FUNCTION "JsonW_LNK_Ack" : Void
{ S7_Optimized_Access := 'TRUE' }
VERSION : 0.1
   VAR_IN_OUT
      Buf : Array[*] of Byte;   // 출력 버퍼
      Pos : DInt;   // 다음 쓸 절대 인덱스 (< 0 = 오류 유지)
      Val : "LNK_Ack";   // 쓸 값
   END_VAR


BEGIN
	// GENERATED by gr-contract gen-link from "LNK_Ack" sig 16#FF5482FF - do not edit
	// wire-spec 2 : 선언 순서, 공백 없음. 버퍼가 모자라면 Pos := LNK_JERR_OVERFLOW (끈끈한 오류, 호출자가 끝에 한 번 확인)
	"Json_WRaw"(Buf := #Buf, Pos := #Pos, Lit := '{"RefType":');
	"Json_WUInt"(Buf := #Buf, Pos := #Pos, Val := #Val.RefType);
	"Json_WRaw"(Buf := #Buf, Pos := #Pos, Lit := ',"RefSeq":');
	"Json_WUInt"(Buf := #Buf, Pos := #Pos, Val := #Val.RefSeq);
	"Json_WRaw"(Buf := #Buf, Pos := #Pos, Lit := ',"Code":');
	"Json_WInt"(Buf := #Buf, Pos := #Pos, Val := #Val.Code);
	"Json_WRaw"(Buf := #Buf, Pos := #Pos, Lit := ',"Text":');
	"Json_WStr"(Buf := #Buf, Pos := #Pos, Val := #Val.Text);
	"Json_WRaw"(Buf := #Buf, Pos := #Pos, Lit := '}');
END_FUNCTION
